FUNCTION GET_SHORTEST_PATH
VAR_INPUT
	nCurrentNode : INT;
	aParents : ARRAY[1..24] OF INT;
END_VAR
VAR
END_VAR

IF NOT (nCurrentNode = 0) THEN
	GET_SHORTEST_PATH(aParents[nCurrentNode], aParents);
	GLOBALS.aRoadFlags[nCurrentNode] := TRUE;
END_IF

END_FUNCTION

(* stored: Version 1.1.0.1, ProductVersion 3.1.4024.12
   POU GET_SHORTEST_PATH: Id {880a5606-6801-48af-8197-1a765a98a14a}, SpecialFunc None *)
